{attribute 'qualified_only'}
{attribute 'strict'}
TYPE E_ACTUATOR_EVENT :
(
	NONE	:= 0,
	
	(* events corresponding to commands *)
	RESET,
	INIT,
	STOP,
	ENABLE,
	DISABLE,
	ON,
	OFF,
	
	(* 
		Events corresponding to internal events 
	*)
	
	INITON,		// Needed for detection of HW failures during initialisation
	INITOFF,
	DISABLEON,
	DISABLEOFF,
	
	(* events mapped to HW signals *)
	ISON,
	ISOFF,

	HWOK,
	ERRHW,
	ERRMAXON,
	ERRTIMEOUT,
	ERRINIT,
	ERRDISABLE
	
);
END_TYPE

(* stored: Version 1.1.0.1, ProductVersion 3.1.4024.3
   DUT E_ACTUATOR_EVENT: Id {b9b752d4-78ea-4bbd-a5f6-5682bd13dc8f} *)
